Fanuc KAREL source: kt00881.KL

-- PROVISIONAL review KL for V1013-1; original PC SHA256 f6a006659f84d2a92009fe44e07f7203dc6f5635dbb91f3fc4d0635ca9e97e6d
-- Incomplete behavior may be omitted. Consult companion uncertainty JSON. Do not deploy.
PROGRAM KT00881
%NOLOCKGROUP
VAR
  I1 : INTEGER
  I2 : INTEGER
  OUT : REAL
BEGIN
  -- UNRESOLVED_PC offsets 5-16; opcodes 2E,23
  -- UNRESOLVED_PC offsets 21-32; opcodes 2E,23
  -- UNRESOLVED_PC offsets 37-48; opcodes 2E,23
  -- UNRESOLVED_PC offsets 53-64; opcodes 2E,23
  -- UNRESOLVED_PC offsets 69-94; opcodes 27,27,21,64,27,21,64,76,23
  -- UNRESOLVED_PC offsets 99-103; opcodes 7F
END KT00881
